Fanuc KAREL source: kt00303.KL

-- PROVISIONAL review KL for V1013-1; original PC SHA256 755615cd21a6e0a9a79ed1437dd2338bf3d26f4f4403b73ee81a3d216f29d07a
-- Incomplete behavior may be omitted. Consult companion uncertainty JSON. Do not deploy.
PROGRAM KT00303
%NOLOCKGROUP
VAR
  I2 : INTEGER
  OUT : BOOLEAN
-- UNRESOLVED_DECL Y1 type=002018
BEGIN
  -- UNRESOLVED_PC offsets 5-19; opcodes 2E,22,9D,33,B2
  -- UNRESOLVED_PC offsets 24-35; opcodes 2E,23
  -- UNRESOLVED_PC offsets 40-62; opcodes 22,9D,33,B1,21,58,23
  -- UNRESOLVED_PC offsets 67-71; opcodes 7F
END KT00303
